(* PLC project  *)

CONFIGURATION raspi4b
END_CONFIGURATION
